{attribute 'GeneratedUsingTerminal: EP1122-0001-0018'}
{attribute addProperty BoxType "EP1122-0001-0018"}
{attribute addProperty Id "A_0027_EP1258_0001_0016EP1258_58F475DD56A_0028_EP1258_0001_0017EP1258_58F475DD56A_0029_EP1258_0001_0018EP1258_58F475DD56A_0030_EP1258_0001_0019EP1258_58F475DD56A_0031_EP1258_0001_0020EP1258_58F475DD56A_0032_EP1258_0002_0016EP1258_58F475DD56A_0033_EP1258_0002_0017EP1258_58F475DD56A_0034_EP1258_0002_0018EP1258_58F475DD56A_0035_EP1258_0002_0019EP1258_58F475DD56A_0036_EP1258_0002_0020EP1258_58F475DD56A_0037_EP1312_0001_0016A_0037_EP1312_0001_0016_211442AD890"}
{attribute addProperty CRC "1942733950"}
{attribute addProperty Size "1450"}
TYPE A_0026_EP1122_0001_0018_73CBC47E EXTENDS EP1122_1FC0878B :
STRUCT
	{attribute addProperty Name "A_0027(EP1258-0001-0016)"}
	{attribute addProperty PreviousPort "A_0026(EP1122-0001-0018) : D"}
	A_0027_EP1258_0001_0016 : EP1258_58F475DD;
	{attribute addProperty Name "A_0028(EP1258-0001-0017)"}
	{attribute addProperty PreviousPort "A_0027(EP1258-0001-0016) : B"}
	A_0028_EP1258_0001_0017 : EP1258_58F475DD;
	{attribute addProperty Name "A_0029(EP1258-0001-0018)"}
	{attribute addProperty PreviousPort "A_0028(EP1258-0001-0017) : B"}
	A_0029_EP1258_0001_0018 : EP1258_58F475DD;
	{attribute addProperty Name "A_0030(EP1258-0001-0019)"}
	{attribute addProperty PreviousPort "A_0029(EP1258-0001-0018) : B"}
	A_0030_EP1258_0001_0019 : EP1258_58F475DD;
	{attribute addProperty Name "A_0031(EP1258-0001-0020)"}
	{attribute addProperty PreviousPort "A_0030(EP1258-0001-0019) : B"}
	A_0031_EP1258_0001_0020 : EP1258_58F475DD;
	{attribute addProperty Name "A_0032(EP1258-0002-0016)"}
	{attribute addProperty PreviousPort "A_0031(EP1258-0001-0020) : B"}
	A_0032_EP1258_0002_0016 : EP1258_58F475DD;
	{attribute addProperty Name "A_0033(EP1258-0002-0017)"}
	{attribute addProperty PreviousPort "A_0032(EP1258-0002-0016) : B"}
	A_0033_EP1258_0002_0017 : EP1258_58F475DD;
	{attribute addProperty Name "A_0034(EP1258-0002-0018)"}
	{attribute addProperty PreviousPort "A_0033(EP1258-0002-0017) : B"}
	A_0034_EP1258_0002_0018 : EP1258_58F475DD;
	{attribute addProperty Name "A_0035(EP1258-0002-0019)"}
	{attribute addProperty PreviousPort "A_0034(EP1258-0002-0018) : B"}
	A_0035_EP1258_0002_0019 : EP1258_58F475DD;
	{attribute addProperty Name "A_0036(EP1258-0002-0020)"}
	{attribute addProperty PreviousPort "A_0035(EP1258-0002-0019) : B"}
	A_0036_EP1258_0002_0020 : EP1258_58F475DD;
	{attribute addProperty Name "A_0037(EP1312-0001-0016)"}
	{attribute addProperty PreviousPort "A_0036(EP1258-0002-0020) : B"}
	A_0037_EP1312_0001_0016 : A_0037_EP1312_0001_0016_211442AD;
END_STRUCT
END_TYPE

(* stored: Version 1.2.0.0, ProductVersion 3.1.4024.11
   DUT A_0026_EP1122_0001_0018_73CBC47E: Id {4adda755-8e0d-4cf5-a771-b7b896fedfde} *)
